// TwinCAT 3 PLC project Untitled1
// ProgramVersion: 3.1.4026.1+c9eadab3edd020c56c333d811d5b3c408c2550c8
// libraries:
//   Tc2_MC2, * (Beckhoff Automation GmbH)
//   Tc2_Standard, * (Beckhoff Automation GmbH)
//   Tc2_System, * (Beckhoff Automation GmbH)
//   Tc3_EventLogger, * (Beckhoff Automation GmbH)
//   TcUnit, * (www.tcunit.org)
// project tree:
//   DUTs/ CONSTANTS.TcGVL, E_AxisEvent.TcDUT, ST_16BIT.TcDUT, ST_AxisParameter.TcDUT
//   Motion Function Block/ FB_Axis.TcPOU, FB_RingBuffer_MCMoveAbsolute.TcPOU, FB_RingBuffer_MCMoveModulo.TcPOU, FB_RingBuffer_MCMoveRelative.TcPOU, FB_RingBuffer_MCMoveVelocity.TcPOU
//   / PlcTask.TcTTO
//   POUs/ MAIN.TcPOU
//   UnitTest/BasicMotionFunction/ FB_Jog_Test.TcPOU, FB_MoveAbsolute_Test.TcPOU, FB_MoveModulo_Test.TcPOU, FB_MoveRelative_Test.TcPOU, FB_MoveVelocity_Test.TcPOU
//   UnitTest/ PRG_Test.TcPOU
// real-time tasks:
//   TASK PlcTask: cycle T#10ms, priority 20, ADS port 350
// motion (NC):
//   TASK NC-Task 1 SAF: cycle T#2ms, priority 4, ADS port 501
//   TASK NC-Task 1 SVB: cycle T#10ms, priority 8, ADS port 511
//   AXIS Axis 1 (id 1)
//   AXIS Axis 2 (id 2)
//   AXIS Axis 3 (id 3)
//   AXIS Axis 4 (id 4)
//     OtherSettings: AllowMotionCmdToSlave=true
//     encoder EncType=1
//     drive DrvType=5
//       Analog: TorqueSetpointScale=10, ScaleFactorActTorque=0.1
//     controller CtrType=1
//       CtrPara: PriorControlFactor=1
//         Observer: BandWidth=20
//   AXIS Axis 5 (id 5)
//     OtherSettings: AllowMotionCmdToSlave=true
//     encoder EncType=1
//     drive DrvType=5
//       Analog: TorqueSetpointScale=10, ScaleFactorActTorque=0.1
//     controller CtrType=1
//       CtrPara: PriorControlFactor=1
//         Observer: BandWidth=20
//   AXIS Axis 6 (id 6)
//     OtherSettings: AllowMotionCmdToSlave=true
//     encoder EncType=1
//     drive DrvType=5
//       Analog: TorqueSetpointScale=10, ScaleFactorActTorque=0.1
//     controller CtrType=1
//       CtrPara: PriorControlFactor=1
//         Observer: BandWidth=20
// variable links:
//   Untitled1 Instance <-> NC-Task 1 SAF/Axes/Axis 1
//     PlcTask Inputs/PRG_Test.fbMoveAbsoluteTest.fbTestAxis._axis.NcToPlc <-> Outputs/ToPlc
//     PlcTask Outputs/PRG_Test.fbMoveAbsoluteTest.fbTestAxis._axis.PlcToNc <-> Inputs/FromPlc
//   Untitled1 Instance <-> NC-Task 1 SAF/Axes/Axis 2
//     PlcTask Inputs/PRG_Test.fbMoveModuloTest.fbTestAxis._axis.NcToPlc <-> Outputs/ToPlc
//     PlcTask Outputs/PRG_Test.fbMoveModuloTest.fbTestAxis._axis.PlcToNc <-> Inputs/FromPlc
//   Untitled1 Instance <-> NC-Task 1 SAF/Axes/Axis 3
//     PlcTask Inputs/PRG_Test.fbMoveVelocity.fbTestAxis._axis.NcToPlc <-> Outputs/ToPlc
//     PlcTask Outputs/PRG_Test.fbMoveVelocity.fbTestAxis._axis.PlcToNc <-> Inputs/FromPlc
//   Untitled1 Instance <-> NC-Task 1 SAF/Axes/Axis 4
//     PlcTask Inputs/PRG_Test.fbMoveRelativeTest.fbTestAxis._axis.NcToPlc <-> Outputs/ToPlc
//     PlcTask Outputs/PRG_Test.fbMoveRelativeTest.fbTestAxis._axis.PlcToNc <-> Inputs/FromPlc
//   Untitled1 Instance <-> NC-Task 1 SAF/Axes/Axis 5
//     PlcTask Inputs/PRG_Test.fbJogTest.fbTestAxis._axis.NcToPlc <-> Outputs/ToPlc
//     PlcTask Outputs/PRG_Test.fbJogTest.fbTestAxis._axis.PlcToNc <-> Inputs/FromPlc
//   Untitled1 Instance <-> NC-Task 1 SAF/Axes/Axis 6
//     PlcTask Inputs/MAIN.axis1._axis.NcToPlc <-> Outputs/ToPlc
//     PlcTask Outputs/MAIN.axis1._axis.PlcToNc <-> Inputs/FromPlc

CONFIGURATION Untitled1
    RESOURCE PLC ON TwinCAT3
        TASK PlcTask(INTERVAL := T#10ms, PRIORITY := 20);
        PROGRAM MAIN WITH PlcTask : MAIN;
        PROGRAM PRG_Test WITH PlcTask : PRG_Test;
    END_RESOURCE
END_CONFIGURATION

// ---- DUTs/E_AxisEvent.TcDUT
TYPE E_AxisEvent :(Enable := 1, Disable:=2, Halt:=3, Reset:=4, MoveAbsolute:=5, MoveModulo := 6, MoveRelative := 7, MoveVelocity := 8, Jog := 9)  UINT;
END_TYPE

// ---- DUTs/ST_16BIT.TcDUT
TYPE ST_16BIT :
STRUCT
	bit1 : BIT;
	bit2 : BIT;
	bit3 : BIT;
	bit4 : BIT;
	bit5: BIT;
	bit6 : BIT;
	bit7 : BIT;
	bit8 : BIT;
	bit9 : BIT;
	bit10 : BIT;
	bit11 : BIT;
	bit12 : BIT;
	bit13 : BIT;
	bit14 : BIT;
	bit15 : BIT;
	bit16 : BIT;
END_STRUCT
END_TYPE

// ---- DUTs/ST_AxisParameter.TcDUT
TYPE ST_AxisParameter :
STRUCT
	Velocity : LREAL;
	Acceleration : LREAL;
	Deceleration : LREAL;
	Jerk : LREAL;
END_STRUCT
END_TYPE

// ---- DUTs/CONSTANTS.TcGVL
{attribute 'qualified_only'}
VAR_GLOBAL CONSTANT
	BASIC_AXIS_ALARM_COUNT		 : UINT := 9; //E
END_VAR

// ---- POUs/MAIN.TcPOU
PROGRAM MAIN
VAR
	axis1 : FB_Axis;
	testStep: INT := 3;
	
	Pos : LREAL;
	Velo : LREAL;
	bButton: BOOL;
	bErrorReset: BOOL;

	Test1_AxisParameter : ST_AxisParameter := (Acceleration := 100, Deceleration := 100, Velocity := 50, Jerk :=500);
	Test2_AxisParameter : ST_AxisParameter := (Acceleration := 1050, Deceleration := 500, Velocity := 150, Jerk :=300);
	Test3_AxisParameter : ST_AxisParameter := (Acceleration := 105, Deceleration := 50, Velocity := 15, Jerk :=30);
	rrTest : LREAL;
END_VAR

axis1.UpdateAxisStatus(); //모터 지령 받기전에 상태 업데이트 필요 (코드 제일 상단에서 콜 해야함 ) 

CASE testStep OF
	1:
		//Do Nothing
	3:
		axis1(stAxisParameter := Test1_AxisParameter); //속도 설정 Test1
	4:
		axis1(stAxisParameter := Test2_AxisParameter); //속도 설정 Test2
	10:
		axis1.Enable(); //서보 온
		testStep := 1;
	20:
		axis1.Disable(); //서보 오프
		testStep := 1;
	30:
		axis1.MoveAbsolute(1000,TRUE); //1000의 절대위치로 이동 , 다른 모션 명령 중지후 바로 실행
		testStep := 1;
	40:
		axis1.MoveAbsolute(-1000, TRUE);// -1000의 절대위치로 이동 , 다른 모션 명령 중지후 바로 실행
		testStep := 1;
	50:
		axis1.MoveAbsolute(2000, FALSE);// 2000의 절대위치로 이동, 다른 모션 명령 실행중일땐 명령 무시
		testStep := 1;
	55:
		axis1.Jog(TRUE, FALSE, E_JOGMODE.MC_JOGMODE_STANDARD_SLOW, 0);
	56:
		axis1.MoveModulo(rrTest, MC_Direction.MC_Negative_Direction, FALSE);
		teststep:=1;
	57:
		axis1.MoveModulo(rrTest, MC_Direction.MC_Positive_Direction, FALSE);
		teststep:=1;
	58:
		axis1.MoveModulo(rrTest, MC_Direction.MC_Shortest_Way, FALSE);
		teststep:=1;
	60:
		axis1.Halt(); // 모션 명령 정지
		testStep := 1;
	70:
		axis1.Reset();
		testStep := 1;
		
		
	//CASE 1 : 500위치로 이동 후 -1000위치로 이동	
	100:
		axis1.MoveAbsolute(500, TRUE); //500 위치로 이동
		testStep := 101;
	101:
		IF axis1.InPosition THEN //500 위치인지 체크
			testStep := 110;
		END_IF
	110:
		axis1.MoveAbsolute(-1000,TRUE); // -1000위치로 이동
		testStep := 111;
	111:
		IF axis1.InPosition THEN // -1000위치인지 체크
			testStep := 1;
		END_IF
		
	//CASE 1 끝


 	//CASE 2 : 10000위치로 이동 중 bButton 신호를 받고 0위치로 이동
	200:
		axis1.MoveAbsolute(10000,TRUE);
		IF bButton THEN
			testStep := 210;
			bButton := FALSE;
		END_IF
	210:
		axis1.MoveAbsolute(0,TRUE);
		IF axis1.InPosition THEN
			testStep := 1;
		END_IF
	//CASE 2 끝
END_CASE

axis1.CyclicLogic(); //펑션 콜 하는 기능 주기적으로 계속 실행되야함

END_PROGRAM

// ---- Motion Function Block/FB_Axis.TcPOU
{attribute 'reflection'}
FUNCTION_BLOCK FB_Axis
VAR_INPUT
	stAxisParameter : ST_AxisParameter;
END_VAR
VAR_OUTPUT
	Error : BOOL;
	ErrorID : UDINT;
	Busy : BOOL;
END_VAR
VAR
	{attribute 'instance-path'}
	{attribute 'noinit'}
	_MyPath : STRING;
	
	_Initalized : BOOL;
	_axis : AXIS_REF;
	MCJog							  : MC_Jog;
	RingBuffer_MCMoveAbsolute : FB_RingBuffer_MCMoveAbsolute;
	RingBuffer_MCMoveRelative : FB_RingBuffer_MCMoveRelative;
	RingBuffer_MCMoveVelocity : FB_RingBuffer_MCMoveVelocity;
	RingBuffer_MCMoveModulo	  : FB_RingBuffer_MCMoveModulo;
	MCMoveAbsolute			  : POINTER TO MC_MoveAbsolute;
	MCMoveRelative			  : POINTER TO MC_MoveRelative;
	MCMoveVelocity			  : POINTER TO MC_MoveVelocity;
	MCMoveModulo			  : POINTER TO MC_MoveModulo;
	MCPower : MC_Power;
	MCHalt: MC_Halt;
	MCReset : MC_Reset;
	AxisAlarm : ARRAY[1..CONSTANTS.BASIC_AXIS_ALARM_COUNT] OF FB_TcMessage;
END_VAR

PROPERTY Axis : REFERENCE TO AXIS_REF
GET
Axis REF= _Axis;
END_GET
END_PROPERTY

METHOD CyclicLogic
VAR_INPUT
END_VAR
IF NOT _Initalized THEN
	Initalize();
	_Initalized := TRUE;
	RETURN;
END_IF

(* MC_Power *)
MCPower(Axis := _Axis);
IF MCPower.Error THEN
	Error	 := TRUE;
	ErrorID := MCPower.ErrorID;
END_IF

(* MC_Halt *)
MCHalt(Axis := _Axis);
IF NOT MCHalt.Busy THEN
	IF MCHalt.Error THEN
		Error	 := TRUE;
		ErrorID := MCHalt.ErrorID;
	ELSE
		MCHalt(Axis := _Axis, Execute := FALSE);
	END_IF
END_IF

(* MC_MoveAbsolute *)
RingBuffer_MCMoveAbsolute(Axis := _Axis);
IF (MCMoveAbsolute <> 0) AND_THEN NOT MCMoveAbsolute^.Busy THEN
	IF MCMoveAbsolute^.Error THEN
		Error	 := TRUE;
		ErrorID := MCMoveAbsolute^.ErrorID;
	ELSE
		MCMoveAbsolute^(Axis := _Axis, Execute := FALSE);
	END_IF
END_IF


(* MC_MoveRelative *)
RingBuffer_MCMoveRelative(Axis := _Axis);
IF (MCMoveRelative <> 0) AND_THEN NOT MCMoveRelative^.Busy THEN
	IF MCMoveRelative^.Error THEN
		Error	 := TRUE;
		ErrorID := MCMoveRelative^.ErrorID;
	ELSE
		MCMoveRelative^(Axis := _Axis, Execute := FALSE);
	END_IF
END_IF

(* MC_MoveVelocity *)
RingBuffer_MCMoveVelocity(Axis := _Axis);
IF (MCMoveVelocity <> 0) AND_THEN ((NOT MCMoveVelocity^.Busy) OR MCMoveVelocity^.InVelocity) THEN
	IF MCMoveVelocity^.Error THEN
		Error	 := TRUE;
		ErrorID := MCMoveVelocity^.ErrorID;
	ELSE
		MCMoveVelocity^(Axis := _Axis, Execute := FALSE);
	END_IF
END_IF

(* MC_MoveModulo *)
RingBuffer_MCMoveModulo(Axis := _Axis);
IF (MCMoveModulo <> 0) AND_THEN NOT MCMoveModulo^.Busy THEN
	IF MCMoveModulo^.Error THEN
		Error	 := TRUE;
		ErrorID := MCMoveModulo^.ErrorID;
	ELSE
		MCMoveModulo^(Axis := _Axis, Execute := FALSE);
	END_IF
END_IF


(*MC_Jog*)
MCJog(Axis := _Axis);
IF MCJog.Error THEN
	Error	 := TRUE;
	ErrorID := MCJog.ErrorID;
END_IF

(* FB_Reset *)
MCReset(Axis := _axis); 
IF NOT MCReset.Busy THEN
	IF MCReset.Error THEN
		Error				:= TRUE;
		ErrorID			   	:= MCReset.ErrorID;
	END_IF
	
	MCReset(Axis := _Axis, Execute := FALSE);
END_IF

Busy := ((MCMoveAbsolute <> 0) AND_THEN MCMoveAbsolute^.Busy) OR ((MCMoveRelative <> 0) AND_THEN MCMoveRelative^.Busy) OR ((MCMoveVelocity <> 0) AND_THEN MCMoveVelocity^.Busy) OR ((MCMoveModulo <> 0) AND_THEN MCMoveModulo^.Busy) OR MCJog.Busy OR MCHalt.Busy OR McReset.Busy;
	 

// _Busy := ((MCMoveAbsolute <> 0) AND_THEN MCMoveAbsolute^.Busy) OR ((MCMoveRelative <> 0) AND_THEN MCMoveRelative^.Busy) OR ((MCMoveVelocity <> 0) AND_THEN MCMoveVelocity^.Busy) OR ((MCMoveModulo <> 0) AND_THEN MCMoveModulo^.Busy) OR MCJog.Busy OR MCHalt.Busy OR ((ipHomeMethod <> 0) AND_THEN ipHomeMethod.Busy) OR ((ipResetMethod <> 0) AND_THEN ipResetMethod.Busy) OR
// 		 ((ipExternalSequence <> 0) AND_THEN ipExternalSequence.Busy) OR MCWriteParameter.Busy OR MCWriteBoolParameter.Busy;
END_METHOD

METHOD Disable : BOOL
VAR_INPUT
END_VAR
MCPower(Axis := _axis, Enable := FALSE, Enable_Positive := FALSE, Enable_Negative := FALSE);
Disable := TRUE;
AxisAlarm[E_AxisEvent.Disable].Send(0);
END_METHOD

METHOD Enable : BOOL
VAR_INPUT
END_VAR
MCPower(Axis := _axis, Enable := TRUE, Enable_Positive := TRUE, Enable_Negative := TRUE);
Enable := TRUE;

AxisAlarm[E_AxisEvent.Enable].Send(0);
END_METHOD

PROPERTY Enabled : BOOL
GET
Enabled := _axis.NcToPlc.stateDword.0;
END_GET
END_PROPERTY

METHOD Halt : BOOL
VAR_INPUT
END_VAR
IF Error AND _Axis.Status.Error THEN
	(* It's possible that a function block errored but
	not the NC itself--in this case we can allow a stop command.
	If the NC axis has a real fault then we want a successful reset first *)
	RETURN;
END_IF

MCHalt(Axis			:= _Axis,
	   Execute		:= TRUE,
	   Deceleration := stAxisParameter.Deceleration,
	   Jerk			:= stAxisParameter.Jerk);

Halt := TRUE;
AxisAlarm[E_AxisEvent.Halt].Send(0);
END_METHOD

METHOD PROTECTED Initalize
AxisAlarm[E_AxisEvent.Disable].CreateEx(stEventEntry := TC_Events.AxisEvents.Disable, 0);
AxisAlarm[E_AxisEvent.Enable].CreateEx(stEventEntry := TC_Events.AxisEvents.Enable, 0);
AxisAlarm[E_AxisEvent.Halt].CreateEx(stEventEntry := TC_Events.AxisEvents.Halt, 0);
AxisAlarm[E_AxisEvent.Reset].CreateEx(stEventEntry := TC_Events.AxisEvents.Reset, 0);
AxisAlarm[E_AxisEvent.MoveAbsolute].CreateEx(stEventEntry := TC_Events.AxisEvents.MoveAbsolute, 0);
AxisAlarm[E_AxisEvent.MoveModulo].CreateEx(stEventEntry := TC_Events.AxisEvents.MoveModulo, 0);
AxisAlarm[E_AxisEvent.MoveRelative].CreateEx(stEventEntry := TC_Events.AxisEvents.MoveRelative, 0);
AxisAlarm[E_AxisEvent.MoveVelocity].CreateEx(stEventEntry := TC_Events.AxisEvents.MoveVelocity, 0);
AxisAlarm[E_AxisEvent.Jog].CreateEx(stEventEntry := TC_Events.AxisEvents.Jog, 0);
END_METHOD

PROPERTY InPosition : BOOL
GET
InPosition := Axis.NcToPLC.stateDword.4;
END_GET
END_PROPERTY

METHOD Jog : BOOL
VAR_INPUT
	JogFW	 : BOOL;
	JogBW	 : BOOL;
	JogMode	 : E_JogMode;
	Position : LREAL;
END_VAR
IF Error THEN
	RETURN;
END_IF

MCJog(Axis		   := _Axis,
	  JogForward   := JogFW,
	  JogBackwards := JogBW,
	  Mode		   := JogMode,
	  Position	   := Position,
	  Velocity	   := stAxisParameter.Velocity,
	  Acceleration := stAxisParameter.Acceleration,
	  Deceleration := stAxisParameter.Deceleration,
	  Jerk		   := stAxisParameter.Jerk);
Jog := TRUE;
END_METHOD

METHOD MoveAbsolute : BOOL
VAR_INPUT
	Position : LREAL;
	AbortPrevious : BOOL;
END_VAR
IF Error THEN
	RETURN;
ELSE
	IF (Busy AND NOT AbortPrevious) THEN
		RETURN;
	END_IF
END_IF

MCMoveAbsolute := RingBuffer_MCMoveAbsolute.GetNewFB();
MCMoveAbsolute^(Axis		 := _Axis,
				Execute		 := TRUE,
				Position	 := Position,
				Velocity	 := stAxisParameter.Velocity,
				Acceleration := stAxisParameter.Acceleration,
				Deceleration := stAxisParameter.Deceleration,
				Jerk		 := stAxisParameter.Jerk);
				
MoveAbsolute := TRUE;
AxisAlarm[E_AxisEvent.MoveAbsolute].Send(0);
END_METHOD

METHOD MoveModulo : BOOL
VAR_INPUT
	Position	  : LREAL;
	Direction	  : MC_Direction;
	AbortPrevious : BOOL;
END_VAR
IF Error THEN
	RETURN;
ELSE
	IF (Busy AND NOT AbortPrevious) THEN
		RETURN;
	END_IF
END_IF

MCMoveModulo := RingBuffer_MCMoveModulo.GetNewFB();
MCMoveModulo^(Axis		   := _Axis,
			  Execute	   := TRUE,
			  Position	   := Position,
			  Velocity	   := stAxisParameter.Velocity,
			  Acceleration := stAxisParameter.Acceleration,
			  Deceleration := stAxisParameter.Deceleration,
			  Jerk		   := stAxisParameter.Jerk,
			  Direction	   := Direction);

MoveModulo := TRUE;
AxisAlarm[E_AxisEvent.MoveModulo].Send(0);
END_METHOD

METHOD MoveRelative : BOOL
VAR_INPUT
	Distance	  : LREAL;
	AbortPrevious : BOOL;
END_VAR
IF Error THEN
	RETURN;
ELSE
	IF (Busy AND NOT AbortPrevious) THEN
		RETURN;
	END_IF
END_IF

MCMoveRelative := RingBuffer_MCMoveRelative.GetNewFB();
MCMoveRelative^(Axis		 := _Axis,
				Execute		 := TRUE,
				Distance	 := Distance,
				Velocity	 := stAxisParameter.Velocity,
				Acceleration := stAxisParameter.Acceleration,
				Deceleration := stAxisParameter.Deceleration,
				Jerk		 := stAxisParameter.Jerk);

MoveRelative := TRUE;
AxisAlarm[E_AxisEvent.MoveRelative].Send(0);
END_METHOD

METHOD MoveVelocity : BOOL
VAR_INPUT
	Velocity	  : LREAL;
	AbortPrevious : BOOL;
END_VAR
IF Error THEN
	RETURN;
ELSE
	IF (Busy AND NOT AbortPrevious) THEN
		RETURN;
	END_IF
END_IF

// IF ABS(Velocity) > _AxisParameters.fVeloMaximum THEN
// 	Trace('Velocity setpoint exceeds axis limit');
// END_IF

IF Velocity < 0 THEN
	MCMoveVelocity			  := RingBuffer_MCMoveVelocity.GetNewFB();
	MCMoveVelocity^.Direction := MC_Negative_Direction;
ELSE
	MCMoveVelocity			  := RingBuffer_MCMoveVelocity.GetNewFB();
	MCMoveVelocity^.Direction := MC_Positive_Direction;
END_IF

 
MCMoveVelocity^(Axis		 := _Axis,
				Execute		 := TRUE,
				Velocity	 := ABS(Velocity),
				Acceleration := stAxisParameter.Acceleration,
				Deceleration := stAxisParameter.Deceleration,
				Jerk		 := stAxisParameter.Jerk);

MoveVelocity := TRUE;
AxisAlarm[E_AxisEvent.MoveVelocity].Send(0);
END_METHOD

METHOD Reset : BOOL;
VAR_INPUT
END_VAR
MCReset(Axis := _Axis, Execute := TRUE);
Busy	 := TRUE;
Error := FALSE;
ErrorID := 0;
Reset := TRUE;

ResetFBs();

AxisAlarm[E_AxisEvent.Reset].Send(0);
Reset := TRUE;
END_METHOD

METHOD PRIVATE ResetFBs
VAR_INPUT
END_VAR
IF MCMoveAbsolute <> 0 THEN
	IF MCMoveAbsolute^.Error THEN
		MCMoveAbsolute^(Axis := _Axis, Execute := FALSE);
	END_IF
END_IF

IF MCMoveRelative <> 0 THEN
	IF MCMoveRelative^.Error THEN
		MCMoveRelative^(Axis := _Axis, Execute := FALSE);
	END_IF
END_IF

IF MCMoveVelocity <> 0 THEN
	IF MCMoveVelocity^.Error THEN
		MCMoveVelocity^(Axis := _Axis, Execute := FALSE);
	END_IF
END_IF

IF MCMoveModulo <> 0 THEN
	IF MCMoveModulo^.Error THEN
		MCMoveModulo^(Axis := _Axis, Execute := FALSE);
	END_IF
END_IF

IF MCJog.Error THEN
	MCJog(Axis := _Axis, JogForward := FALSE, JogBackwards := FALSE);
END_IF

IF MCHalt.Error THEN
	MCHalt(Axis := _Axis, Execute := FALSE);
END_IF

//    IF MCMoveSuperimposed.Error THEN

//        MCMoveSuperimposed(Axis := _Axis, Execute := FALSE);

//    END_IF

//    IF MCAbortSuperposition.Error THEN

//        MCAbortSuperposition(Axis := _Axis, Execute := FALSE);

// //    END_IF  

(* Temperaly delete It could be used *)
// IF MCReadParameterSet.Error THEN
// 	MCReadParameterSet(Axis := _Axis, Parameter := _AxisParameters, Execute := FALSE);
// END_IF
// 
// IF MCWriteBoolParameter.Error THEN
// 	MCWriteBoolParameter(Axis := _Axis, Execute := FALSE);
// END_IF
// 
// IF MCWriteParameter.Error THEN
// 	MCWriteParameter(Axis := _Axis, Execute := FALSE);
// END_IF
END_METHOD

METHOD UpdateAxisStatus
Axis.ReadStatus(); //Axis 상태 업데이트
END_METHOD

END_FUNCTION_BLOCK

// ---- Motion Function Block/FB_RingBuffer_MCMoveAbsolute.TcPOU
FUNCTION_BLOCK FB_RingBuffer_MCMoveAbsolute
VAR_IN_OUT
	Axis: AXIS_REF;
END_VAR
VAR
	MCMoveAbsolute: ARRAY[0..1] OF MC_MoveAbsolute;
	_CurrentFB: UDINT;
	i: UDINT;
END_VAR

FOR i := 0 TO 1 DO
	MCMoveAbsolute[i](Axis := Axis);
END_FOR

PROPERTY CurrentFB : POINTER TO MC_MoveAbsolute
GET
CurrentFB := ADR(MCMoveAbsolute[_CurrentFB]);
END_GET
END_PROPERTY

METHOD GetNewFB : POINTER TO MC_MoveAbsolute
_CurrentFB := _CurrentFB + 1;
IF _CurrentFB > 1 THEN
	MCMoveAbsolute[1].Execute := FALSE;
	_CurrentFB				  := 0;
ELSE
	MCMoveAbsolute[_CurrentFB - 1].Execute := FALSE;
END_IF

GetNewFB := ADR(MCMoveAbsolute[_CurrentFB]);
END_METHOD

END_FUNCTION_BLOCK

// ---- Motion Function Block/FB_RingBuffer_MCMoveRelative.TcPOU
FUNCTION_BLOCK FB_RingBuffer_MCMoveRelative
VAR_IN_OUT
	Axis : AXIS_REF;
END_VAR

VAR_OUTPUT
END_VAR

VAR
	MCMoveRelative : ARRAY[0..1] OF MC_MoveRelative;
	_CurrentFB	   : UDINT;
	i			   : UDINT;
END_VAR

(* This buffer ensures you always have a clean FB to use for a move *)

FOR i := 0 TO 1 DO
	MCMoveRelative[i](Axis := Axis);
END_FOR

PROPERTY CurrentFB : POINTER TO MC_MoveRelative
GET
CurrentFB := ADR(MCMoveRelative[_CurrentFB]);
END_GET
END_PROPERTY

METHOD GetNewFB : POINTER TO MC_MoveRelative
VAR_INPUT
END_VAR
_CurrentFB := _CurrentFB + 1;
IF _CurrentFB > 1 THEN
	MCMoveRelative[1].Execute := FALSE;
	_CurrentFB				  := 0;
ELSE
	MCMoveRelative[_CurrentFB - 1].Execute := FALSE;
END_IF

GetNewFB := ADR(MCMoveRelative[_CurrentFB]);
END_METHOD

END_FUNCTION_BLOCK

// ---- Motion Function Block/FB_RingBuffer_MCMoveVelocity.TcPOU
FUNCTION_BLOCK FB_RingBuffer_MCMoveVelocity
VAR_IN_OUT
	Axis : AXIS_REF;
END_VAR

VAR_OUTPUT
END_VAR

VAR
	MCMoveVelocity : ARRAY[0..1] OF MC_MoveVelocity;
	_CurrentFB	   : UDINT;
	i			   : UDINT;
END_VAR

(* This buffer ensures you always have a clean FB to use for a move *)

FOR i := 0 TO 1 DO
	MCMoveVelocity[i](Axis := Axis);
END_FOR

PROPERTY CurrentFB : POINTER TO MC_MoveVelocity
GET
CurrentFB := ADR(MCMoveVelocity[_CurrentFB]);
END_GET
END_PROPERTY

METHOD GetNewFB : POINTER TO MC_MoveVelocity
VAR_INPUT
END_VAR
_CurrentFB := _CurrentFB + 1;
IF _CurrentFB > 1 THEN
	MCMoveVelocity[1].Execute := FALSE;
	_CurrentFB				  := 0;
ELSE
	MCMoveVelocity[_CurrentFB - 1].Execute := FALSE;
END_IF

GetNewFB := ADR(MCMoveVelocity[_CurrentFB]);
END_METHOD

END_FUNCTION_BLOCK

// ---- Motion Function Block/FB_RingBuffer_MCMoveModulo.TcPOU
FUNCTION_BLOCK FB_RingBuffer_MCMoveModulo
VAR_IN_OUT
	Axis : AXIS_REF;
END_VAR

VAR_OUTPUT
END_VAR

VAR
	MCMoveModulo : ARRAY[0..1] OF MC_MoveModulo;
	_CurrentFB	 : UDINT;
	i			 : UDINT;
END_VAR

(* This buffer ensures you always have a clean FB to use for a move *)

FOR i := 0 TO 1 DO
	MCMoveModulo[i](Axis := Axis);
END_FOR

PROPERTY CurrentFB : POINTER TO MC_MoveModulo
GET
CurrentFB := ADR(MCMoveModulo[_CurrentFB]);
END_GET
END_PROPERTY

METHOD GetNewFB : POINTER TO MC_MoveModulo
VAR_INPUT
END_VAR
_CurrentFB := _CurrentFB + 1;
IF _CurrentFB > 1 THEN
	MCMoveModulo[1].Execute := FALSE;
	_CurrentFB				:= 0;
ELSE
	MCMoveModulo[_CurrentFB - 1].Execute := FALSE;
END_IF

GetNewFB := ADR(MCMoveModulo[_CurrentFB]);
END_METHOD

END_FUNCTION_BLOCK

// ---- UnitTest/PRG_Test.TcPOU
PROGRAM PRG_Test
VAR
	fbMoveAbsoluteTest : FB_MoveAbsolute_Test;
	fbMoveModuloTest : FB_MoveModulo_Test;
	fbMoveVelocity : FB_MoveVelocity_Test;
	fbMoveRelativeTest : FB_MoveRelative_Test;
	fbJogTest : FB_Jog_Test;
END_VAR

(* UnitTest *)
RUN();

END_PROGRAM

// ---- UnitTest/BasicMotionFunction/FB_MoveAbsolute_Test.TcPOU
FUNCTION_BLOCK FB_MoveAbsolute_Test EXTENDS TcUnit.FB_TestSuite

VAR
	fbTestAxis : FB_Axis;
	stAxisParameter : ST_AxisParameter := (Acceleration := 1000, Deceleration := 1000, Jerk := 2000, Velocity := 1000);

END_VAR

MoveAbsolute1000();
MoveAbsolute100();
MoveAbsolute1000_negDir();

METHOD MoveAbsolute100
VAR_INST
	step: INT;
	
	fbTon : TON := (PT:= T#10s);
	EXPECTED_RESULT : INT := 20;
END_VAR
IF TEST_ORDERED('MoveAbsolute100') THEN
		
	fbTestAxis.CyclicLogic();
	CASE step OF
		0:
			fbTestAxis.stAxisParameter := stAxisParameter;
			fbTestAxis.Enable();
			IF fbTestAxis.Enabled THEN
				step := 10;
			END_IF
		10:
			IF fbTestAxis.MoveAbsolute(100,FALSE) = TRUE THEN
				step := 11;
			END_IF
			
		11:
			IF NOT fbTestAxis.Busy AND fbTestAxis.InPosition THEN
				step := 20;
			END_IF
		
		20: //Done
		
	
	END_CASE
	fbTestAxis.CyclicLogic();
	
	
	fbTon(IN := TRUE);
	IF fbTon.Q OR step = 20 THEN
		AssertEquals(Expected := EXPECTED_RESULT, Actual := step, Message := 'MoveAbsolute100 didnt work');
		TEST_FINISHED();
	END_IF
END_IF
END_METHOD

METHOD MoveAbsolute1000
VAR_INST
	step: INT;
	
	fbTon : TON := (PT:= T#10s);
	EXPECTED_RESULT : INT := 20;
END_VAR
IF TEST_ORDERED('MoveAbsolute1000') THEN
		
	
	fbTestAxis.CyclicLogic();
	CASE step OF
		0:
			fbTestAxis.stAxisParameter := stAxisParameter;
			fbTestAxis.Enable();
			IF fbTestAxis.Enabled THEN
				step := 10;
			END_IF
		10:
			IF fbTestAxis.MoveAbsolute(1000,FALSE) = TRUE THEN
				step := 11;
			END_IF
			
		11:
			IF NOT fbTestAxis.Busy AND fbTestAxis.InPosition THEN
				step := 20;
			END_IF
		20: //Done
	END_CASE
	
	fbTestAxis.CyclicLogic();
	
	
	fbTon(IN := TRUE);
	IF fbTon.Q OR step = 20 THEN
		AssertEquals(Expected := EXPECTED_RESULT, Actual := step, Message := 'MoveAbsolute1000 didnt work');
		TEST_FINISHED();
	END_IF
END_IF
END_METHOD

METHOD MoveAbsolute1000_negDir
VAR_INST
	step: INT;
	
	fbTon : TON := (PT:= T#10s);
	EXPECTED_RESULT : INT := 20;
END_VAR
IF TEST_ORDERED('MoveAbsolute1000_negDir') THEN
		
	fbTestAxis.CyclicLogic();
	CASE step OF
		0:
			fbTestAxis.stAxisParameter := stAxisParameter;
			fbTestAxis.Enable();
			IF fbTestAxis.Enabled THEN
				step := 10;
			END_IF
		10:
			IF fbTestAxis.MoveAbsolute(-1000,FALSE) = TRUE THEN
				step := 11;
			END_IF
			
		11:
			IF NOT fbTestAxis.Busy AND fbTestAxis.InPosition THEN
				step := 20;
			END_IF
		20: //Done
	END_CASE
	
	fbTestAxis.CyclicLogic();
	
	
	fbTon(IN := TRUE);
	IF fbTon.Q OR step = 20 THEN
		AssertEquals(Expected := EXPECTED_RESULT, Actual := step, Message := 'MoveAbsolute1000_negDir');
		TEST_FINISHED();
	END_IF
END_IF
END_METHOD

END_FUNCTION_BLOCK

// ---- UnitTest/BasicMotionFunction/FB_MoveModulo_Test.TcPOU
FUNCTION_BLOCK FB_MoveModulo_Test EXTENDS TcUnit.FB_TestSuite

VAR
	fbTestAxis : FB_Axis;
	stAxisParameter : ST_AxisParameter := (Acceleration := 1000, Deceleration := 1000, Jerk := 2000, Velocity := 1000);

END_VAR

MoveModulo100_posDir();
MoveModulo1000_negDir();
MoveModulo150_Shortestway();

//현재 위치보다 작은 각도를 목표로 움직이고 target pos이 360를 넘으면 한바퀴 더 돌게됨

METHOD MoveModulo100_posDir
VAR_INST
	step: INT;
	
	fbTon : TON := (PT:= T#10s);
	EXPECTED_RESULT : INT := 20;
END_VAR
IF TEST_ORDERED('MoveAbsolute100') THEN
		
	fbTestAxis.CyclicLogic();
	CASE step OF
		0:
			fbTestAxis.stAxisParameter := stAxisParameter;
			fbTestAxis.Enable();
			IF fbTestAxis.Enabled THEN
				step := 10;
			END_IF
		10:
			IF fbTestAxis.MoveModulo(100, MC_Direction.MC_Positive_Direction, FALSE) = TRUE THEN
				step := 11;
			END_IF
			
		11:
			IF NOT fbTestAxis.Busy AND fbTestAxis.InPosition THEN
				step := 20;
			END_IF
		
		20: //Done
		
	
	END_CASE
	fbTestAxis.CyclicLogic();
	
	
	fbTon(IN := TRUE);
	IF fbTon.Q OR step = 20 THEN
		AssertEquals(Expected := EXPECTED_RESULT, Actual := step , Message := 'MoveModulo100 didnt work');
		TEST_FINISHED();
	END_IF
END_IF
END_METHOD

METHOD MoveModulo1000_negDir
VAR_INST
	step: INT;
	
	fbTon : TON := (PT:= T#10s);
	EXPECTED_RESULT : int := 20;
END_VAR
IF TEST_ORDERED('MoveAbsolute1000_negDir') THEN
		
	fbTestAxis.CyclicLogic();
	CASE step OF
		0:
			fbTestAxis.stAxisParameter := stAxisParameter;
			fbTestAxis.Enable();
			IF fbTestAxis.Enabled THEN
				step := 10;
			END_IF
		10:
			IF fbTestAxis.MoveModulo(1000, MC_Direction.MC_Negative_Direction, FALSE) = TRUE THEN
				step := 11;
			END_IF
			
		11:
			IF NOT fbTestAxis.Busy AND fbTestAxis.InPosition THEN
				step := 20;
			END_IF
		20: //Done
	END_CASE
	
	fbTestAxis.CyclicLogic();
	
	
	fbTon(IN := TRUE);
	IF fbTon.Q OR step = 20 THEN
		AssertEquals(Expected := EXPECTED_RESULT, Actual := step, Message := 'MoveAbsolute1000_negDir');
		TEST_FINISHED();
	END_IF
END_IF
END_METHOD

METHOD MoveModulo150_Shortestway
VAR_INST
	step: INT;
	
	fbTon : TON := (PT:= T#10s);
	EXPECTED_RESULT : INT := 20;
END_VAR
IF TEST_ORDERED('MoveModulo150') THEN
		
	
	fbTestAxis.CyclicLogic();
	CASE step OF
		0:
			fbTestAxis.stAxisParameter := stAxisParameter;
			fbTestAxis.Enable();
			IF fbTestAxis.Enabled THEN
				step := 10;
			END_IF
		10:
			IF fbTestAxis.MoveModulo(150,MC_Direction.MC_Shortest_Way,FALSE) = TRUE THEN
				step := 11;
			END_IF
			
		11:
			IF NOT fbTestAxis.Busy AND fbTestAxis.InPosition THEN
				step := 20;
			END_IF
		20: //Done
	END_CASE
	
	fbTestAxis.CyclicLogic();
	
	
	fbTon(IN := TRUE);
	IF fbTon.Q OR step = 20 THEN
		AssertEquals(Expected := EXPECTED_RESULT, Actual := step, Message := 'MoveModulo150_shortest way didnt work');
		TEST_FINISHED();
	END_IF
END_IF
END_METHOD

END_FUNCTION_BLOCK

// ---- UnitTest/BasicMotionFunction/FB_MoveVelocity_Test.TcPOU
FUNCTION_BLOCK FB_MoveVelocity_Test EXTENDS TcUnit.FB_TestSuite

VAR
	fbTestAxis : FB_Axis;
	stAxisParameter : ST_AxisParameter := (Acceleration := 1000, Deceleration := 1000, Jerk := 2000, Velocity := 1000);

END_VAR

MoveAbsolute1000();
MoveVelocity100();
MoveAbsolute1000_negDir();

METHOD MoveAbsolute1000
VAR_INST
	step: INT;
	
	fbTon : TON := (PT:= T#10s);
	EXPECTED_RESULT : INT := 20;
END_VAR
IF TEST_ORDERED('MoveVelocity1000') THEN
		
	fbTestAxis.CyclicLogic();
	CASE step OF
		0:
			fbTestAxis.stAxisParameter := stAxisParameter;
			fbTestAxis.Enable();
			IF fbTestAxis.Enabled THEN
				step := 10;
			END_IF
		10:
			IF fbTestAxis.MoveVelocity(1000,TRUE) = TRUE THEN
				step := 11;
			END_IF
			
		11:
			IF fbTestAxis.Axis.NcToPlc.ActVelo >= 999 THEN
				step := 20;
			END_IF
		
		20: //Done
		
	
	END_CASE
	fbTestAxis.CyclicLogic();
	
	
	fbTon(IN := TRUE);
	IF fbTon.Q OR step = 20 THEN
		AssertEquals(Expected := EXPECTED_RESULT, Actual := step, Message := 'MoveVelocity1000 didnt work');
		TEST_FINISHED();
	END_IF
END_IF
END_METHOD

METHOD MoveAbsolute1000_negDir
VAR_INST
	step: INT;
	
	fbTon : TON := (PT:= T#10s);
	EXPECTED_RESULT : INT := 20;
END_VAR
IF TEST_ORDERED('MoveVelocity1000_negDir') THEN
		
	fbTestAxis.CyclicLogic();
	CASE step OF
		0:
			fbTestAxis.stAxisParameter := stAxisParameter;
			fbTestAxis.Enable();
			IF fbTestAxis.Enabled THEN
				step := 10;
			END_IF
		10:
			IF fbTestAxis.MoveVelocity(-1000,TRUE) = TRUE THEN
				step := 11;
			END_IF
			
		11:
			IF fbTestAxis.Axis.NcToPlc.ActVelo <= -999 THEN
				step := 20;
				fbTestAxis.Halt();
			END_IF
		
		20: 
			
			//Done
		
	
	END_CASE
	fbTestAxis.CyclicLogic();
	
	
	fbTon(IN := TRUE);
	IF fbTon.Q OR step = 20 THEN
		AssertEquals(Expected := EXPECTED_RESULT, Actual := step, Message := 'MoveVelocity100 didnt work');
		TEST_FINISHED();
	END_IF
END_IF
END_METHOD

METHOD MoveVelocity100
VAR_INST
	step: INT;
	
	fbTon : TON := (PT:= T#10s);
	EXPECTED_RESULT : INT := 20;
END_VAR
IF TEST_ORDERED('MoveVelocity100') THEN
		
	fbTestAxis.CyclicLogic();
	CASE step OF
		0:
			fbTestAxis.stAxisParameter := stAxisParameter;
			fbTestAxis.Enable();
			IF fbTestAxis.Enabled THEN
				step := 10;
			END_IF
		10:
			IF fbTestAxis.MoveVelocity(100,FALSE) = TRUE THEN
				step := 11;
			END_IF
			
		11:
			IF fbTestAxis.Axis.NcToPlc.ActVelo >= 99 THEN
				step := 20;
			END_IF
		
		20: //Done
		
	
	END_CASE
	fbTestAxis.CyclicLogic();
	
	
	fbTon(IN := TRUE);
	IF fbTon.Q OR step = 20 THEN
		AssertEquals(Expected := EXPECTED_RESULT, Actual := step, Message := 'MoveVelocity100 didnt work');
		TEST_FINISHED();
	END_IF
END_IF
END_METHOD

END_FUNCTION_BLOCK

// ---- UnitTest/BasicMotionFunction/FB_MoveRelative_Test.TcPOU
FUNCTION_BLOCK FB_MoveRelative_Test EXTENDS TcUnit.FB_TestSuite
VAR
	fbTestAxis : FB_Axis;
	stAxisParameter : ST_AxisParameter := (Acceleration := 1000, Deceleration := 1000, Jerk := 2000, Velocity := 1000);
END_VAR

MoveRelative1000();
MoveRelative200();
MoveRelative1300_negDir();

METHOD MoveRelative1000
VAR_INST
	step : INT;
	fbTon : TON;
	EXPECTED_RESULT : INT := 20;
END_VAR
TEST_ORDERED('MoveRelative1000');

fbTon(IN := TRUE, PT := T#10S);
fbTestAxis.CyclicLogic();

CASE step OF
	0:
		fbTestAxis(stAxisParameter := stAxisParameter);
		fbTestAxis.Enable();
		IF fbTestAxis.Enabled THEN
			step := 10;
		END_IF
	10:
		IF fbTestAxis.MoveRelative(1000, FALSE) THEN
			step := 11;
		END_IF
	11:
		IF NOT fbTestAxis.Busy AND fbTestAxis.InPosition THEN
			step := 20;
		END_IF
	20:
	
END_CASE
IF fbTon.Q OR step = 20 THEN
	AssertEquals(EXPECTED_RESULT, step, 'relative1000');
	TEST_FINISHED();
END_IF
END_METHOD

METHOD MoveRelative1300_negDir
VAR_INST
	step : INT;
	fbTon : TON;
	EXPECTED_RESULT : INT := 20;
END_VAR
TEST_ORDERED('MoveRelative1300_negDir');

fbTon(IN := TRUE, PT := T#10S);
fbTestAxis.CyclicLogic();

CASE step OF
	0:
		fbTestAxis(stAxisParameter := stAxisParameter);
		fbTestAxis.Enable();
		IF fbTestAxis.Enabled THEN
			step := 10;
		END_IF
	10:
		IF fbTestAxis.MoveRelative(-1300, FALSE) THEN
			step := 11;
		END_IF
	11:
		IF NOT fbTestAxis.Busy AND fbTestAxis.InPosition THEN
			step := 20;
		END_IF
	20:
	
END_CASE
IF fbTon.Q OR step = 20 THEN
	AssertEquals(EXPECTED_RESULT, step, 'MoveRelative1300_negDir');
	TEST_FINISHED();
END_IF
END_METHOD

METHOD MoveRelative200
VAR_INST
	step : INT;
	fbTon : TON;
	EXPECTED_RESULT : INT := 20;
END_VAR
TEST_ORDERED('MoveRelative200');

fbTon(IN := TRUE, PT := T#10S);
fbTestAxis.CyclicLogic();

CASE step OF
	0:
		fbTestAxis(stAxisParameter := stAxisParameter);
		fbTestAxis.Enable();
		IF fbTestAxis.Enabled THEN
			step := 10;
		END_IF
	10:
		IF fbTestAxis.MoveRelative(200, FALSE) THEN
			step := 11;
		END_IF
	11:
		IF NOT fbTestAxis.Busy AND fbTestAxis.InPosition THEN
			step := 20;
		END_IF
	20:
	
END_CASE
IF fbTon.Q OR step = 20 THEN
	AssertEquals(EXPECTED_RESULT, step, 'relative1000');
	TEST_FINISHED();
END_IF
END_METHOD

END_FUNCTION_BLOCK

// ---- UnitTest/BasicMotionFunction/FB_Jog_Test.TcPOU
FUNCTION_BLOCK FB_Jog_Test EXTENDS TcUnit.FB_TestSuite

VAR
	fbTestAxis : FB_Axis;
	stAxisParameter : ST_AxisParameter := (Acceleration := 1000, Deceleration := 1000, Jerk := 2000, Velocity := 1000);

END_VAR

JogBackword();
JogForward();
MoveBackAndForth();
//JOG커멘드는 중간에 콜이 안되면 마지막에 지령준 방향으로 계쏙감

METHOD JogBackword
VAR_INST
	step: INT;
	
	fbTon : TON := (PT:= T#10s);
	EXPECTED_RESULT : INT := 20;
END_VAR
IF TEST_ORDERED('JogBackword') THEN		
	fbTestAxis.CyclicLogic();
	CASE step OF
		0:
			fbTestAxis.stAxisParameter := stAxisParameter;
			fbTestAxis.Enable();
			IF fbTestAxis.Enabled THEN
				step := 10;
			END_IF
		10:
			fbTestAxis.Jog(FALSE, TRUE,E_JogMode.MC_JOGMODE_STANDARD_FAST,1000);
			IF fbTestAxis.Axis.NcToPlc.ActPos <= -100 THEN
				step := 20;
				fbTestAxis.Jog(FALSE, FALSE,E_JogMode.MC_JOGMODE_STANDARD_FAST,0);
			END_IF
		
		20: //Done
		
	
	END_CASE
	fbTestAxis.CyclicLogic();
	
	
	fbTon(IN := TRUE);
	IF fbTon.Q OR step = 20 THEN
		AssertEquals(Expected := EXPECTED_RESULT, Actual := step, Message := 'JogBackward');
		TEST_FINISHED();
	END_IF
END_IF
END_METHOD

METHOD JogForward
VAR_INST
	step: INT;
	
	fbTon : TON := (PT:= T#10s);
	EXPECTED_RESULT : INT := 20;
END_VAR
IF TEST_ORDERED('JogForward') THEN
	fbTestAxis.CyclicLogic();
	CASE step OF
		0:
			fbTestAxis.stAxisParameter := stAxisParameter;
			fbTestAxis.Enable();
			IF fbTestAxis.Enabled THEN
				step := 10;
			END_IF
		10:
			fbTestAxis.Jog(TRUE, FALSE,E_JogMode.MC_JOGMODE_STANDARD_FAST,0);
			IF fbTestAxis.Axis.NcToPlc.ActPos >= 1000 THEN
				step := 20;
				fbTestAxis.Jog(FALSE, FALSE,E_JogMode.MC_JOGMODE_STANDARD_FAST,0);
			END_IF
			
		
		
		20: //Done
		
	
	END_CASE
	fbTestAxis.CyclicLogic();
	
	
	fbTon(IN := TRUE);
	IF fbTon.Q OR step = 20 THEN
		AssertEquals(Expected := EXPECTED_RESULT, Actual := step, Message := 'JogForward');
		TEST_FINISHED();
	END_IF
END_IF
END_METHOD

METHOD MoveBackAndForth
VAR_INST
	step: INT;
	
	fbTon : TON := (PT:= T#10s);
	EXPECTED_RESULT : INT := 20;
END_VAR
IF TEST_ORDERED('MoveBackAndForth') THEN
		
	fbTestAxis.CyclicLogic();
	CASE step OF
		0:
			fbTestAxis.stAxisParameter := stAxisParameter;
			fbTestAxis.Enable();
			IF fbTestAxis.Enabled THEN
				step := 10;
			END_IF
		10:
			fbTestAxis.Jog(TRUE, FALSE,E_JogMode.MC_JOGMODE_STANDARD_FAST,0);
			IF fbTestAxis.Axis.NcToPlc.ActPos >= 1000 THEN
				step := 15;
			END_IF
		15:
			fbTestAxis.Jog(FALSE, TRUE,E_JogMode.MC_JOGMODE_STANDARD_FAST,0);
			IF fbTestAxis.Axis.NcToPlc.ActPos <= -100 THEN
				step := 20;
				fbTestAxis.Jog(FALSE, FALSE,E_JogMode.MC_JOGMODE_STANDARD_FAST,0);
			END_IF
		
		20: //Done
		
	
	END_CASE
	fbTestAxis.CyclicLogic();
	
	
	fbTon(IN := TRUE);
	IF fbTon.Q OR step = 20 THEN
		AssertEquals(Expected := EXPECTED_RESULT, Actual := step, Message := 'MoveBackAndForth');
		TEST_FINISHED();
	END_IF
END_IF
END_METHOD

END_FUNCTION_BLOCK
